{attribute 'linkalways'} 
{attribute 'no_explicit_call' := 'This FB is a CLASS and must be accessed using methods or properties'}
{attribute 'enable_dynamic_creation'}
FUNCTION_BLOCK _Array0to1OfINT EXTENDS ArrayDatatypeBase
VAR CONSTANT
	lBound : DINT := 0;
	uBound : DINT := 1;
END_VAR
VAR
	localData : ARRAY [lBound..uBound] OF INT;
	activeData : REFERENCE TO ARRAY [lBound..uBound] OF INT REF= localData;
	elements : ARRAY [lBound..uBound] OF _INT(0);
	baseType : _INT(0);
END_VAR

PROPERTY PUBLIC Address : PVOID
GET
Address := ADR(activeData);
END_GET
END_PROPERTY

PROPERTY PUBLIC BaseDatatype : I_Datatype
GET
BaseDatatype := baseType;
END_GET
END_PROPERTY

METHOD PUBLIC ClearReference
VAR_INPUT
END_VAR
activeData REF= localData;
SetElementReference();
END_METHOD

METHOD PUBLIC Clone : I_Datatype
VAR
    pClone : POINTER TO _Array0to1OfINT;
END_VAR
pClone := __NEW(_Array0to1OfINT());
pClone^.Value := Value;
Clone := pClone^;
END_METHOD

METHOD FB_init : BOOL
VAR_INPUT
	bInitRetains : BOOL; // if TRUE, the retain variables are initialized (warm start / cold start)
	bInCopyCode : BOOL;  // if TRUE, the instance afterwards gets moved into the copy code (online change)
END_VAR
SetElementReference();
END_METHOD

METHOD PUBLIC GetElementAsDatatypeByIndex : I_Datatype
VAR_INPUT
	Index : DINT;
END_VAR
GetElementAsDatatypeByIndex := elements[Index];
END_METHOD

METHOD PUBLIC GetElementByIndex : REFERENCE TO _INT;
VAR_INPUT
	Index : DINT;
END_VAR
GetElementByIndex REF= elements[Index];
END_METHOD

PROPERTY PUBLIC LowerBound : DINT
GET
LowerBound := lBound;
END_GET
END_PROPERTY

METHOD PUBLIC MakeReferenceTo
VAR_INPUT
	ReferenceTarget : REFERENCE TO ARRAY [lBound..uBound] OF INT;
END_VAR
activeData REF= ReferenceTarget;
SetElementReference();
END_METHOD

METHOD PROTECTED OnSerializeArrayValues
VAR_INPUT
	Serializer : I_Serializer;
END_VAR
VAR
	i : DINT;
END_VAR
FOR i := lBound TO uBound DO
	elements[i].SerializeWith(Serializer);
END_FOR
END_METHOD

METHOD PROTECTED SetElementReference
VAR_INPUT
END_VAR
VAR
	i : DINT;
END_VAR
FOR i := lBound TO uBound DO
	elements[i].MakeReferenceTo(activeData[i]);
END_FOR
END_METHOD

PROPERTY PUBLIC Size : UDINT
GET
Size := SIZEOF(activeData);
END_GET
END_PROPERTY

METHOD PROTECTED TryDeserializeArrayValues : BOOL
VAR_INPUT
	Deserializer : I_Deserializer;
	Feedback : I_DeserializerFeedback;
END_VAR
VAR
	enumerator : I_DeserializerArrayForwardEnumerator;
	i : DINT;
END_VAR
enumerator := Deserializer.GetArrayEnumerator();
i := lBound;

WHILE enumerator.MoveNext() AND i <= uBound DO
	
	IF NOT elements[i].TryDeserializeFrom(enumerator.Current, Feedback) THEN
		EXIT;
	END_IF
	i := i + 1;

END_WHILE
enumerator.Dispose();
END_METHOD

METHOD TryMakeReferenceTo : BOOL
VAR_INPUT
	Target : I_Datatype;
END_VAR
VAR
	targetAsArray : I_ArrayDatatype;
	pTargetData : POINTER TO ARRAY [lBound..uBound] OF INT;
END_VAR
IF NOT Target.TryResolveAsArrayDatatype(targetAsArray) THEN
	RETURN;
END_IF

IF NOT (targetAsArray.Identifier = Identifier) THEN
	RETURN;
END_IF

pTargetData := Target.Address;
activeData REF= pTargetData^;
SetElementReference();
TryMakeReferenceTo := TRUE;
END_METHOD

PROPERTY PUBLIC UpperBound : DINT
GET
UpperBound := ubound;
END_GET
END_PROPERTY

PROPERTY PUBLIC Value : REFERENCE TO ARRAY [lBound..uBound] OF INT;
GET
Value ref= activeData;
END_GET
END_PROPERTY

END_FUNCTION_BLOCK

(* stored: Version 1.1.0.1, ProductVersion 3.1.4024.13
   POU _Array0to1OfINT: Id {8703c02d-48ab-0f77-2e76-a0923efb1581}, SpecialFunc None
   Folder Core: Id {e4e1ccd1-7627-0c6c-1c39-b63cd7e9133d}
   Folder Constructor: Id {4e612049-0702-08c5-1e96-46459b86ea4b}
   Folder Protected: Id {00e406fa-a1ef-0cc9-05a2-c0837dba8a06}
   Folder Customize: Id {7d0803fb-15e9-0e7f-3c73-d89ddc3c3826}
   Property Address: Id {36fb73b9-52b1-0055-0993-3bf86b81dc3d}
   Get Get: Id {ebcb375b-848e-0f55-1367-f53b188e8b67}
   Property BaseDatatype: Id {476ae6ae-89b4-0350-3c68-37fd26cbb10a}
   Get Get: Id {5c69cf4f-36c2-0f1d-2a44-ce7f612f9d58}
   Method ClearReference: Id {bb19a876-480d-023d-37c6-d1be642c2f67}
   Method Clone: Id {23fbbab2-ee98-0911-3684-8bf1b28e1251}
   Method FB_init: Id {bf3f6501-f765-0c0f-2af9-30c8967d44be}
   Method GetElementAsDatatypeByIndex: Id {2b197645-1160-0e61-2c8c-a724abf805d1}
   Method GetElementByIndex: Id {0a69e9a4-e5d7-0c2c-09c8-836eace6cb66}
   Property LowerBound: Id {115df441-73a4-06fb-343e-21c593f29022}
   Get Get: Id {86911fc5-f78c-0250-0794-dc620bfa6fcf}
   Method MakeReferenceTo: Id {2ab78e00-74e9-0632-0fbf-861c7b27ce26}
   Method OnSerializeArrayValues: Id {79a10b82-8729-0934-25c9-896671625568}
   Method SetElementReference: Id {c14ce1c6-1ea5-020a-20e1-0d127673adbf}
   Property Size: Id {53609e23-a4d7-0ffd-2bde-217f4755c159}
   Get Get: Id {3bded9bd-eb92-04da-1bf5-dabfe54e904d}
   Method TryDeserializeArrayValues: Id {27b499ee-29c3-0eb0-21d1-975c73b9add4}
   Method TryMakeReferenceTo: Id {b5423845-94f1-0111-0650-5e12eed9a98c}
   Property UpperBound: Id {51be9716-b3ba-08be-0460-0f78795a590a}
   Get Get: Id {7a1a7281-1e68-06af-160a-a1073871f01e}
   Property Value: Id {cb44f7ee-d84c-017c-3314-5f496a6450b2}
   Get Get: Id {a763e221-5782-029c-2591-db0f7a9de99a} *)
